{attribute 'GeneratedUsingTerminal: ELX1054-0000-0016'}
{attribute addProperty BoxType "ELX1054-0000-0016"}
{attribute addProperty Id "ChannelAT %I*ARRAY[0..3] OF BOOL4"}
{attribute addProperty CRC "1364972313"}
{attribute addProperty Size "4"}
TYPE Input_Type_NC_5EE69541 :
STRUCT
	{attribute addProperty Name "Channel"}
	Channel AT %I* : ARRAY[0..3] OF BOOL;
END_STRUCT
END_TYPE

(* stored: Version 1.2.0.0, ProductVersion 3.1.4024.9
   DUT Input_Type_NC_5EE69541: Id {5e5e69e3-524e-478d-a94b-b1afd2b3e6ec} *)
